// Mitsubishi GX Works2 project: test_backup   PLC: Q02/Q02H

// task Task_01 (event TRUE, interval 0, priority 31): POU_01

PROGRAM POU_01
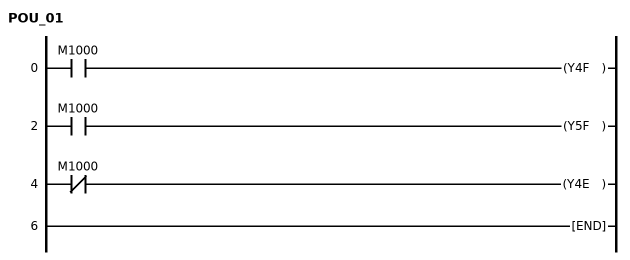
0     LD      M1000
      OUT     Y4F
2     LD      M1000
      OUT     Y5F
4     LDI     M1000
      OUT     Y4E
6     END
END_PROGRAM
